    LOCAL CONST Robtarget Tr_meulage_bavure_258 := [[-0.894256591796875,91.7996015625,80.2160234375],[0.00347787918573702,-0.00302620431421481,0.656413988017704,-0.754386785925172],[0,0,0,0],[8.999999E+09,8.999999E+09,8.999999E+09,8.999999E+09,8.999999E+09,8.999999E+09]];
    LOCAL CONST Robtarget Tr_meulage_bavure_259 := [[-3.09170532226563,91.8315234375,80.2122734375],[0.00491374660901085,-0.00426989771840249,0.655908883103524,-0.754812003172727],[0,0,0,0],[8.999999E+09,8.999999E+09,8.999999E+09,8.999999E+09,8.999999E+09,8.999999E+09]];
    LOCAL CONST Robtarget Tr_meulage_bavure_260 := [[-8.3219912109375,91.974546875,80.1954765625],[0.00744982146467277,-0.00646558456435395,0.655423726856519,-0.755196950900821],[0,0,0,0],[8.999999E+09,8.999999E+09,8.999999E+09,8.999999E+09,8.999999E+09,8.999999E+09]];
    LOCAL CONST Robtarget Tr_meulage_bavure_261 := [[-9.6864931640625,91.992796875,80.193328125],[0.0113222387628506,-0.00981492756750365,0.654945437900396,-0.755527595445528],[0,0,0,0],[8.999999E+09,8.999999E+09,8.999999E+09,8.999999E+09,8.999999E+09,8.999999E+09]];
    LOCAL CONST Robtarget Tr_meulage_bavure_262 := [[-20.53646875,92.018953125,80.1902578125],[0.0166484079195255,-0.0144163975754932,0.65445477578378,-0.755780354632543],[0,0,0,0],[8.999999E+09,8.999999E+09,8.999999E+09,8.999999E+09,8.999999E+09,8.999999E+09]];
    LOCAL CONST Robtarget Tr_meulage_bavure_263 := [[-23.421142578125,92.016859375,80.1905],[0.0234300908490705,-0.020268509523459,0.653923705596549,-0.755925926016153],[0,0,0,0],[8.999999E+09,8.999999E+09,8.999999E+09,8.999999E+09,8.999999E+09,8.999999E+09]];
    LOCAL CONST Robtarget Tr_meulage_bavure_264 := [[-24.027587890625,92.04446875,80.1872578125],[0.0314797870413223,-0.0272072091200353,0.65333054540363,-0.755928560925123],[0,0,0,0],[8.999999E+09,8.999999E+09,8.999999E+09,8.999999E+09,8.999999E+09,8.999999E+09]];
    LOCAL CONST Robtarget Tr_meulage_bavure_265 := [[-26.45446875,92.1919921875,80.1699296875],[0.0404076636865339,-0.0348943430759381,0.652653550089562,-0.755773080423077],[0,0,0,0],[8.999999E+09,8.999999E+09,8.999999E+09,8.999999E+09,8.999999E+09,8.999999E+09]];
    LOCAL CONST Robtarget Tr_meulage_bavure_266 := [[-29.448517578125,92.303890625,80.15678125],[0.0496986305677145,-0.0428854622432543,0.651895870964166,-0.755461883001219],[0,0,0,0],[8.999999E+09,8.999999E+09,8.999999E+09,8.999999E+09,8.999999E+09,8.999999E+09]];
    LOCAL CONST Robtarget Tr_meulage_bavure_267 := [[-31.056060546875,92.1032109375,80.180359375],[0.0587225353541234,-0.0506383751390462,0.651088055954158,-0.755030967708409],[0,0,0,0],[8.999999E+09,8.999999E+09,8.999999E+09,8.999999E+09,8.999999E+09,8.999999E+09]];
    LOCAL CONST Robtarget Tr_meulage_bavure_268 := [[-35.77227734375,91.4953671875,80.251765625],[0.0668827998283126,-0.0576408748993466,0.650281395904972,-0.754545112480257],[0,0,0,0],[8.999999E+09,8.999999E+09,8.999999E+09,8.999999E+09,8.999999E+09,8.999999E+09]];
    LOCAL CONST Robtarget Tr_meulage_bavure_269 := [[-37.007875,91.1575078125,80.291453125],[0.0736958342973869,-0.0634793616298069,0.649541115383601,-0.754079328771524],[0,0,0,0],[8.999999E+09,8.999999E+09,8.999999E+09,8.999999E+09,8.999999E+09,8.999999E+09]];
    LOCAL CONST Robtarget Tr_meulage_bavure_270 := [[-38.72647265625,90.3674296875,80.384265625],[0.0789467515956599,-0.0679716715014017,0.648916433938356,-0.753694052020133],[0,0,0,0],[8.999999E+09,8.999999E+09,8.999999E+09,8.999999E+09,8.999999E+09,8.999999E+09]];
    LOCAL CONST Robtarget Tr_meulage_bavure_271 := [[-42.73101953125,88.3123828125,80.6256796875],[0.0827631719069685,-0.0712303856006982,0.648423147243865,-0.753408197235359],[0,0,0,0],[8.999999E+09,8.999999E+09,8.999999E+09,8.999999E+09,8.999999E+09,8.999999E+09]];
    LOCAL CONST Robtarget Tr_meulage_bavure_272 := [[-44.1032109375,87.88778125,80.6755546875],[0.0855847486840602,-0.0736356000993471,0.648035678832561,-0.753195066467325],[0,0,0,0],[8.999999E+09,8.999999E+09,8.999999E+09,8.999999E+09,8.999999E+09,8.999999E+09]];
    LOCAL CONST Robtarget Tr_meulage_bavure_273 := [[-46.86541796875,86.68584375,80.81675],[0.0882152360556618,-0.0758798732341398,0.647682492084163,-0.752972580120461],[0,0,0,0],[8.999999E+09,8.999999E+09,8.999999E+09,8.999999E+09,8.999999E+09,8.999999E+09]];
    LOCAL CONST Robtarget Tr_meulage_bavure_274 := [[-49.034421875,86.5238125,80.8357890625],[0.0916871696125905,-0.0788508623278929,0.647253511204557,-0.752621350130298],[0,0,0,0],[8.999999E+09,8.999999E+09,8.999999E+09,8.999999E+09,8.999999E+09,8.999999E+09]];
    LOCAL CONST Robtarget Tr_meulage_bavure_275 := [[-53.57986328125,85.9536640625,80.902765625],[0.0972011976752642,-0.0835810818582939,0.646606172682112,-0.751975124173189],[0,0,0,0],[8.999999E+09,8.999999E+09,8.999999E+09,8.999999E+09,8.999999E+09,8.999999E+09]];
    LOCAL CONST Robtarget Tr_meulage_bavure_276 := [[-59.01324609375,86.3367734375,80.8577578125],[0.106067029700948,-0.0911960835370439,0.645540805269948,-0.750806318759605],[0,0,0,0],[8.999999E+09,8.999999E+09,8.999999E+09,8.999999E+09,8.999999E+09,8.999999E+09]];
    LOCAL CONST Robtarget Tr_meulage_bavure_277 := [[-61.2616875,86.3511640625,80.8560703125],[0.119501918726964,-0.10274216646515,0.643784911960041,-0.748801926936105],[0,0,0,0],[8.999999E+09,8.999999E+09,8.999999E+09,8.999999E+09,8.999999E+09,8.999999E+09]];
    LOCAL CONST Robtarget Tr_meulage_bavure_278 := [[-69.158140625,86.6093671875,80.825734375],[0.13852846594866,-0.119099643075277,0.640958292885336,-0.745518347140276],[0,0,0,0],[8.999999E+09,8.999999E+09,8.999999E+09,8.999999E+09,8.999999E+09,8.999999E+09]];
    LOCAL CONST Robtarget Tr_meulage_bavure_279 := [[-70.97525,86.6130703125,80.8253046875],[0.163876976589741,-0.140896368891585,0.636531382818664,-0.740351503317128],[0,0,0,0],[8.999999E+09,8.999999E+09,8.999999E+09,8.999999E+09,8.999999E+09,8.999999E+09]];
    LOCAL CONST Robtarget Tr_meulage_bavure_280 := [[-73.90365625,86.3363203125,80.8578125],[0.195657464814664,-0.168229660305411,0.629881023434704,-0.732575480187997],[0,0,0,0],[8.999999E+09,8.999999E+09,8.999999E+09,8.999999E+09,8.999999E+09,8.999999E+09]];
    LOCAL CONST Robtarget Tr_meulage_bavure_281 := [[-75.0881328125,86.0497421875,80.8914765625],[0.233090996505808,-0.200432374900431,0.620418372993561,-0.721509870266323],[0,0,0,0],[8.999999E+09,8.999999E+09,8.999999E+09,8.999999E+09,8.999999E+09,8.999999E+09]];
    LOCAL CONST Robtarget Tr_meulage_bavure_282 := [[-77.5441015625,85.085125,81.004796875],[0.274367163117045,-0.235949651903377,0.607840699423548,-0.706809808713824],[0,0,0,0],[8.999999E+09,8.999999E+09,8.999999E+09,8.999999E+09,8.999999E+09,8.999999E+09]];
    LOCAL CONST Robtarget Tr_meulage_bavure_283 := [[-78.4228515625,84.0872265625,81.1220234375],[0.316761155122173,-0.272440578103132,0.592433930974092,-0.688810960597378],[0,0,0,0],[8.999999E+09,8.999999E+09,8.999999E+09,8.999999E+09,8.999999E+09,8.999999E+09]];
    LOCAL CONST Robtarget Tr_meulage_bavure_284 := [[-79.9829375,82.004625,81.366671875],[0.357317508371397,-0.307363032722583,0.575147348147079,-0.668623729945487],[0,0,0,0],[8.999999E+09,8.999999E+09,8.999999E+09,8.999999E+09,8.999999E+09,8.999999E+09]];
    LOCAL CONST Robtarget Tr_meulage_bavure_285 := [[-80.3374296875,79.783875,81.627546875],[0.393613708380539,-0.33863296716412,0.557372094713365,-0.647867509726626],[0,0,0,0],[8.999999E+09,8.999999E+09,8.999999E+09,8.999999E+09,8.999999E+09,8.999999E+09]];
    LOCAL CONST Robtarget Tr_meulage_bavure_286 := [[-80.412265625,79.58646875,81.6507421875],[0.424278534863153,-0.365066131411498,0.540492222763307,-0.628158102457493],[0,0,0,0],[8.999999E+09,8.999999E+09,8.999999E+09,8.999999E+09,8.999999E+09,8.999999E+09]];
    LOCAL CONST Robtarget Tr_meulage_bavure_287 := [[-80.42434375,79.4588359375,81.665734375],[0.448961364969328,-0.38635898724885,0.525548437863281,-0.610703909596448],[0,0,0,0],[8.999999E+09,8.999999E+09,8.999999E+09,8.999999E+09,8.999999E+09,8.999999E+09]];
    LOCAL CONST Robtarget Tr_meulage_bavure_288 := [[-80.630734375,75.5483203125,82.125109375],[0.467989879490766,-0.402790192772944,0.513130058558757,-0.596190469819536],[0,0,0,0],[8.999999E+09,8.999999E+09,8.999999E+09,8.999999E+09,8.999999E+09,8.999999E+09]];
    LOCAL CONST Robtarget Tr_meulage_bavure_289 := [[-80.5011015625,72.5830859375,82.4734453125],[0.482071863396728,-0.414965340552088,0.503399466828588,-0.584807200244994],[0,0,0,0],[8.999999E+09,8.999999E+09,8.999999E+09,8.999999E+09,8.999999E+09,8.999999E+09]];
    LOCAL CONST Robtarget Tr_meulage_bavure_290 := [[-80.316984375,68.9543203125,82.8997265625],[0.49206179036456,-0.423611707299164,0.4962002859683,-0.576379729091237],[0,0,0,0],[8.999999E+09,8.999999E+09,8.999999E+09,8.999999E+09,8.999999E+09,8.999999E+09]];
    LOCAL CONST Robtarget Tr_meulage_bavure_291 := [[-80.258484375,65.9367109375,83.25421875],[0.498791013906897,-0.429448562893376,0.491208022376699,-0.570522685813033],[0,0,0,0],[8.999999E+09,8.999999E+09,8.999999E+09,8.999999E+09,8.999999E+09,8.999999E+09]];
    LOCAL CONST Robtarget Tr_meulage_bavure_292 := [[-80.1468203125,54.898046875,84.5509609375],[0.503007913688158,-0.43312019155188,0.488021045124207,-0.566767499026741],[0,0,0,0],[8.999999E+09,8.999999E+09,8.999999E+09,8.999999E+09,8.999999E+09,8.999999E+09]];
    LOCAL CONST Robtarget Tr_meulage_bavure_293 := [[-80.2864375,48.8831328125,85.2575546875],[0.505447763460853,-0.435251867230867,0.486156431674502,-0.564562037712402],[0,0,0,0],[8.999999E+09,8.999999E+09,8.999999E+09,8.999999E+09,8.999999E+09,8.999999E+09]];
    LOCAL CONST Robtarget Tr_meulage_bavure_294 := [[-80.335140625,46.1458203125,85.579109375],[0.50671707315682,-0.436369685524733,0.485181965999149,-0.56339840716462],[0,0,0,0],[8.999999E+09,8.999999E+09,8.999999E+09,8.999999E+09,8.999999E+09,8.999999E+09]];
    LOCAL CONST Robtarget Tr_meulage_bavure_295 := [[-80.3631015625,45.63105078125,85.6395859375],[0.507275210539017,-0.436864892405638,0.484752927928074,-0.56288144881597],[0,0,0,0],[8.999999E+09,8.999999E+09,8.999999E+09,8.999999E+09,8.999999E+09,8.999999E+09]];
    LOCAL CONST Robtarget Tr_meulage_bavure_296 := [[-80.6398046875,44.21337109375,85.806125],[0.507430369539302,-0.437006893390196,0.484634589770416,-0.562733249059194],[0,0,0,0],[8.999999E+09,8.999999E+09,8.999999E+09,8.999999E+09,8.999999E+09,8.999999E+09]];
    !
    !Declaration des points de tronconnage

    !
    !Cycle
    LOCAL PROC Cycle()
        !
        Prise;
        !
        Meulage;
        !
        !
        Depose;
        !
    ENDPROC

    !Trajectoire de prise de la pièce
    LOCAL PROC PRISE()

		!
        !Trigger localisation
        LocalisationPieceTable 703 \model:=1;
        !
        !Approche
		MoveJ Reltool(PicKPosition,0,0,-100),V1000,Z0,Tool_Prehenseur1 \Wobj:=Wobj_vision;
		MoveL Reltool(PicKPosition,0,0,-50),V500,Z0,Tool_Prehenseur1 \Wobj:=Wobj_vision;
		MoveL Reltool(PicKPosition,0,0,-10),V200,Z0,Tool_Prehenseur1 \Wobj:=Wobj_vision;
		MoveL PicKPosition,V100,Fine,Tool_Prehenseur1 \Wobj:=Wobj_vision;

        !Fermeture pince
		Gripper_Close;
        !
		MoveL Reltool(PicKPosition,0,0,-100),V500,Z0,Tool_Prehenseur1 \Wobj:=Wobj_vision;

        !Trigger relocalisation
		LocalisationPiecePrehenseur 703 \model:=1,Ref;
        !
        PEO;
        !
    ENDPROC

    !Trajectoire de tronconnage
    LOCAL PROC Tronconnage()
        !
        !StartMotor1();
        !
        ConfJ \Off;
        ConfL \Off;


    ENDPROC


    !Trajectoire de meulage
    LOCAL PROC Meulage()
        !
        !StartMotor2();
        !

        ConfJ \Off;
        ConfL \Off;


        !---------- Meulage zone : 1 ------------

        !Approche PLAN

        Go_to_Meulage_Plan;
		Tool := ToolOffset(Tool_M1_D500_S0 \Z);

        !
        !Approche
        MoveJ Reltool(Tr_meulage_motif_1_0,0,0,-200),V1000,Z0,Tool \Wobj:=Wobj_Part_0;
        MoveL Reltool(Tr_meulage_motif_1_0,0,0,-100),V500,Z0,Tool \Wobj:=Wobj_Part_0;
        MoveL Reltool(Tr_meulage_motif_1_0,0,0,-10),V100,Z0,Tool \Wobj:=Wobj_Part_0;
        !
        !Trajectoire
        Movel Tr_meulage_motif_1_0,VitesseLente,Z0,Tool \Wobj:=Wobj_Part_0;
        Movel Tr_meulage_motif_1_1,VitesseLente,Z0,Tool \Wobj:=Wobj_Part_0;
        Movel Tr_meulage_motif_1_2,VitesseLente,Z0,Tool \Wobj:=Wobj_Part_0;
        Movel Tr_meulage_motif_1_3,VitesseLente,Z0,Tool \Wobj:=Wobj_Part_0;
        Movel Tr_meulage_motif_1_4,VitesseLente,Z0,Tool \Wobj:=Wobj_Part_0;
        Movel Tr_meulage_motif_1_5,VitesseLente,Z0,Tool \Wobj:=Wobj_Part_0;
        Movel Tr_meulage_motif_1_6,VitesseLente,Z0,Tool \Wobj:=Wobj_Part_0;
        Movel Tr_meulage_motif_1_7,VitesseLente,Z0,Tool \Wobj:=Wobj_Part_0;
        Movel Tr_meulage_motif_1_8,VitesseLente,Z0,Tool \Wobj:=Wobj_Part_0;
        Movel Tr_meulage_motif_1_9,VitesseLente,Z0,Tool \Wobj:=Wobj_Part_0;
        Movel Tr_meulage_motif_1_10,VitesseLente,Z0,Tool \Wobj:=Wobj_Part_0;
        Movel Tr_meulage_motif_1_11,VitesseLente,Z0,Tool \Wobj:=Wobj_Part_0;
        Movel Tr_meulage_motif_1_12,VitesseLente,Z0,Tool \Wobj:=Wobj_Part_0;
        Movel Tr_meulage_motif_1_13,VitesseLente,Z0,Tool \Wobj:=Wobj_Part_0;
        Movel Tr_meulage_motif_1_14,VitesseLente,Z0,Tool \Wobj:=Wobj_Part_0;
        Movel Tr_meulage_motif_1_15,VitesseLente,Z0,Tool \Wobj:=Wobj_Part_0;
        Movel Tr_meulage_motif_1_16,VitesseLente,Z0,Tool \Wobj:=Wobj_Part_0;
        Movel Tr_meulage_motif_1_17,VitesseLente,Z0,Tool \Wobj:=Wobj_Part_0;
        Movel Tr_meulage_motif_1_18,VitesseLente,Z0,Tool \Wobj:=Wobj_Part_0;
        Movel Tr_meulage_motif_1_19,VitesseLente,Z0,Tool \Wobj:=Wobj_Part_0;
        Movel Tr_meulage_motif_1_20,VitesseLente,Z0,Tool \Wobj:=Wobj_Part_0;
        Movel Tr_meulage_motif_1_21,VitesseLente,Z0,Tool \Wobj:=Wobj_Part_0;
        Movel Tr_meulage_motif_1_22,VitesseLente,Z0,Tool \Wobj:=Wobj_Part_0;
        Movel Tr_meulage_motif_1_23,VitesseLente,Z0,Tool \Wobj:=Wobj_Part_0;
        Movel Tr_meulage_motif_1_24,VitesseLente,Z0,Tool \Wobj:=Wobj_Part_0;
        Movel Tr_meulage_motif_1_25,VitesseLente,Z0,Tool \Wobj:=Wobj_Part_0;
        Movel Tr_meulage_motif_1_26,VitesseLente,Z0,Tool \Wobj:=Wobj_Part_0;
        Movel Tr_meulage_motif_1_27,VitesseLente,Z0,Tool \Wobj:=Wobj_Part_0;
        Movel Tr_meulage_motif_1_28,VitesseLente,Z0,Tool \Wobj:=Wobj_Part_0;
        Movel Tr_meulage_motif_1_29,VitesseLente,Z0,Tool \Wobj:=Wobj_Part_0;
        Movel Tr_meulage_motif_1_30,VitesseLente,Z0,Tool \Wobj:=Wobj_Part_0;
        Movel Tr_meulage_motif_1_31,VitesseLente,Z0,Tool \Wobj:=Wobj_Part_0;
        Movel Tr_meulage_motif_1_32,VitesseLente,Z0,Tool \Wobj:=Wobj_Part_0;
        Movel Tr_meulage_motif_1_33,VitesseLente,Z0,Tool \Wobj:=Wobj_Part_0;
        Movel Tr_meulage_motif_1_34,VitesseLente,Z0,Tool \Wobj:=Wobj_Part_0;
        Movel Tr_meulage_motif_1_35,VitesseLente,Z0,Tool \Wobj:=Wobj_Part_0;
        Movel Tr_meulage_motif_1_36,VitesseLente,Z0,Tool \Wobj:=Wobj_Part_0;
        Movel Tr_meulage_motif_1_37,VitesseLente,Z0,Tool \Wobj:=Wobj_Part_0;
        Movel Tr_meulage_motif_1_38,VitesseLente,Z0,Tool \Wobj:=Wobj_Part_0;
        Movel Tr_meulage_motif_1_39,VitesseLente,Z0,Tool \Wobj:=Wobj_Part_0;
        Movel Tr_meulage_motif_1_40,VitesseLente,Z0,Tool \Wobj:=Wobj_Part_0;
        Movel Tr_meulage_motif_1_41,VitesseLente,Z0,Tool \Wobj:=Wobj_Part_0;
        Movel Tr_meulage_motif_1_42,VitesseLente,Z0,Tool \Wobj:=Wobj_Part_0;
        Movel Tr_meulage_motif_1_43,VitesseLente,Z0,Tool \Wobj:=Wobj_Part_0;
        Movel Tr_meulage_motif_1_44,VitesseLente,Z0,Tool \Wobj:=Wobj_Part_0;
        Movel Tr_meulage_motif_1_45,VitesseLente,Z0,Tool \Wobj:=Wobj_Part_0;
        Movel Tr_meulage_motif_1_46,VitesseLente,Z0,Tool \Wobj:=Wobj_Part_0;
        Movel Tr_meulage_motif_1_47,VitesseLente,Z0,Tool \Wobj:=Wobj_Part_0;
        Movel Tr_meulage_motif_1_48,VitesseLente,Z0,Tool \Wobj:=Wobj_Part_0;
        Movel Tr_meulage_motif_1_49,VitesseLente,Z0,Tool \Wobj:=Wobj_Part_0;
        Movel Tr_meulage_motif_1_50,VitesseLente,Z0,Tool \Wobj:=Wobj_Part_0;
        Movel Tr_meulage_motif_1_51,VitesseLente,Z0,Tool \Wobj:=Wobj_Part_0;
        Movel Tr_meulage_motif_1_52,VitesseLente,Z0,Tool \Wobj:=Wobj_Part_0;
        Movel Tr_meulage_motif_1_53,VitesseLente,Z0,Tool \Wobj:=Wobj_Part_0;
        Movel Tr_meulage_motif_1_54,VitesseLente,Z0,Tool \Wobj:=Wobj_Part_0;
        Movel Tr_meulage_motif_1_55,VitesseLente,Z0,Tool \Wobj:=Wobj_Part_0;
        Movel Tr_meulage_motif_1_56,VitesseLente,Z0,Tool \Wobj:=Wobj_Part_0;
        Movel Tr_meulage_motif_1_57,VitesseLente,Z0,Tool \Wobj:=Wobj_Part_0;
        Movel Tr_meulage_motif_1_58,VitesseLente,Z0,Tool \Wobj:=Wobj_Part_0;
        Movel Tr_meulage_motif_1_59,VitesseLente,Z0,Tool \Wobj:=Wobj_Part_0;
        Movel Tr_meulage_motif_1_60,VitesseLente,Z0,Tool \Wobj:=Wobj_Part_0;
        Movel Tr_meulage_motif_1_61,VitesseLente,Z0,Tool \Wobj:=Wobj_Part_0;
        Movel Tr_meulage_motif_1_62,VitesseLente,Z0,Tool \Wobj:=Wobj_Part_0;
        Movel Tr_meulage_motif_1_63,VitesseLente,Z0,Tool \Wobj:=Wobj_Part_0;
        Movel Tr_meulage_motif_1_64,VitesseLente,Z0,Tool \Wobj:=Wobj_Part_0;
        Movel Tr_meulage_motif_1_65,VitesseLente,Z0,Tool \Wobj:=Wobj_Part_0;
        Movel Tr_meulage_motif_1_66,VitesseLente,Z0,Tool \Wobj:=Wobj_Part_0;
        Movel Tr_meulage_motif_1_67,VitesseLente,Z0,Tool \Wobj:=Wobj_Part_0;
        Movel Tr_meulage_motif_1_68,VitesseLente,Z0,Tool \Wobj:=Wobj_Part_0;
        Movel Tr_meulage_motif_1_69,VitesseLente,Z0,Tool \Wobj:=Wobj_Part_0;
        Movel Tr_meulage_motif_1_70,VitesseLente,Z0,Tool \Wobj:=Wobj_Part_0;
        Movel Tr_meulage_motif_1_71,VitesseLente,Z0,Tool \Wobj:=Wobj_Part_0;
        Movel Tr_meulage_motif_1_72,VitesseLente,Z0,Tool \Wobj:=Wobj_Part_0;
        Movel Tr_meulage_motif_1_73,VitesseLente,Z0,Tool \Wobj:=Wobj_Part_0;
        Movel Tr_meulage_motif_1_74,VitesseLente,Z0,Tool \Wobj:=Wobj_Part_0;
        Movel Tr_meulage_motif_1_75,VitesseLente,Z0,Tool \Wobj:=Wobj_Part_0;
        Movel Tr_meulage_motif_1_76,VitesseLente,Z0,Tool \Wobj:=Wobj_Part_0;
        Movel Tr_meulage_motif_1_77,VitesseLente,Z0,Tool \Wobj:=Wobj_Part_0;
        Movel Tr_meulage_motif_1_78,VitesseLente,Z0,Tool \Wobj:=Wobj_Part_0;
        Movel Tr_meulage_motif_1_79,VitesseLente,Z0,Tool \Wobj:=Wobj_Part_0;
        Movel Tr_meulage_motif_1_80,VitesseLente,Z0,Tool \Wobj:=Wobj_Part_0;
        Movel Tr_meulage_motif_1_81,VitesseLente,Z0,Tool \Wobj:=Wobj_Part_0;
        Movel Tr_meulage_motif_1_82,VitesseLente,Z0,Tool \Wobj:=Wobj_Part_0;
        Movel Tr_meulage_motif_1_83,VitesseLente,Z0,Tool \Wobj:=Wobj_Part_0;
        Movel Tr_meulage_motif_1_84,VitesseLente,Z0,Tool \Wobj:=Wobj_Part_0;
        Movel Tr_meulage_motif_1_85,VitesseLente,Z0,Tool \Wobj:=Wobj_Part_0;
        Movel Tr_meulage_motif_1_86,VitesseLente,Z0,Tool \Wobj:=Wobj_Part_0;
        Movel Tr_meulage_motif_1_87,VitesseLente,Z0,Tool \Wobj:=Wobj_Part_0;
        Movel Tr_meulage_motif_1_88,VitesseLente,Z0,Tool \Wobj:=Wobj_Part_0;
        Movel Tr_meulage_motif_1_89,VitesseLente,Z0,Tool \Wobj:=Wobj_Part_0;
        Movel Tr_meulage_motif_1_90,VitesseLente,Z0,Tool \Wobj:=Wobj_Part_0;
        Movel Tr_meulage_motif_1_91,VitesseLente,Z0,Tool \Wobj:=Wobj_Part_0;
        Movel Tr_meulage_motif_1_92,VitesseLente,Z0,Tool \Wobj:=Wobj_Part_0;
        Movel Tr_meulage_motif_1_93,VitesseLente,Z0,Tool \Wobj:=Wobj_Part_0;
        Movel Tr_meulage_motif_1_94,VitesseLente,Z0,Tool \Wobj:=Wobj_Part_0;
        Movel Tr_meulage_motif_1_95,VitesseLente,Z0,Tool \Wobj:=Wobj_Part_0;
        Movel Tr_meulage_motif_1_96,VitesseLente,Z0,Tool \Wobj:=Wobj_Part_0;
        Movel Tr_meulage_motif_1_97,VitesseLente,Z0,Tool \Wobj:=Wobj_Part_0;
        Movel Tr_meulage_motif_1_98,VitesseLente,Z0,Tool \Wobj:=Wobj_Part_0;
        Movel Tr_meulage_motif_1_99,VitesseLente,Z0,Tool \Wobj:=Wobj_Part_0;
        Movel Tr_meulage_motif_1_100,VitesseLente,Z0,Tool \Wobj:=Wobj_Part_0;
        Movel Tr_meulage_motif_1_101,VitesseLente,Z0,Tool \Wobj:=Wobj_Part_0;
        Movel Tr_meulage_motif_1_102,VitesseLente,Z0,Tool \Wobj:=Wobj_Part_0;
        Movel Tr_meulage_motif_1_103,VitesseLente,Z0,Tool \Wobj:=Wobj_Part_0;
        Movel Tr_meulage_motif_1_104,VitesseLente,Z0,Tool \Wobj:=Wobj_Part_0;
        Movel Tr_meulage_motif_1_105,VitesseLente,Z0,Tool \Wobj:=Wobj_Part_0;
        Movel Tr_meulage_motif_1_106,VitesseLente,Z0,Tool \Wobj:=Wobj_Part_0;
        Movel Tr_meulage_motif_1_107,VitesseLente,Z0,Tool \Wobj:=Wobj_Part_0;
        Movel Tr_meulage_motif_1_108,VitesseLente,Z0,Tool \Wobj:=Wobj_Part_0;
        Movel Tr_meulage_motif_1_109,VitesseLente,Z0,Tool \Wobj:=Wobj_Part_0;
        Movel Tr_meulage_motif_1_110,VitesseLente,Z0,Tool \Wobj:=Wobj_Part_0;
        Movel Tr_meulage_motif_1_111,VitesseLente,Z0,Tool \Wobj:=Wobj_Part_0;
        Movel Tr_meulage_motif_1_112,VitesseLente,Z0,Tool \Wobj:=Wobj_Part_0;
        Movel Tr_meulage_motif_1_113,VitesseLente,Z0,Tool \Wobj:=Wobj_Part_0;
        Movel Tr_meulage_motif_1_114,VitesseLente,Z0,Tool \Wobj:=Wobj_Part_0;
        Movel Tr_meulage_motif_1_115,VitesseLente,Z0,Tool \Wobj:=Wobj_Part_0;
        !
        !Degagement
        MoveL Reltool(Tr_meulage_motif_1_115,0,0,-10),V100,Z0,Tool \Wobj:=Wobj_Part_0;
        MoveL Reltool(Tr_meulage_motif_1_115,0,0,-100),V500,Z0,Tool \Wobj:=Wobj_Part_0;
        MoveJ Reltool(Tr_meulage_motif_1_115,0,0,-200),V1000,Z0,Tool \Wobj:=Wobj_Part_0;


        Go_to_Meulage_Plan;
        !
        !

        !---------- Meulage zone : 2 ------------

        !Approche PLAN

        Go_to_Meulage_Plan;
		Tool := ToolOffset(Tool_M1_D500_S0 \Z);

        !
        !Approche
        MoveJ Reltool(Tr_meulage_bavure_0,0,0,-200),V1000,Z0,Tool \Wobj:=Wobj_Part_0;
        MoveL Reltool(Tr_meulage_bavure_0,0,0,-100),V500,Z0,Tool \Wobj:=Wobj_Part_0;
        MoveL Reltool(Tr_meulage_bavure_0,0,0,-10),V100,Z0,Tool \Wobj:=Wobj_Part_0;
        !
        !Trajectoire
        Movel Tr_meulage_bavure_0,VitesseRapide,Z0,Tool \Wobj:=Wobj_Part_0;
        Movel Tr_meulage_bavure_1,VitesseRapide,Z0,Tool \Wobj:=Wobj_Part_0;
        Movel Tr_meulage_bavure_2,VitesseRapide,Z0,Tool \Wobj:=Wobj_Part_0;
        Movel Tr_meulage_bavure_3,VitesseRapide,Z0,Tool \Wobj:=Wobj_Part_0;
        Movel Tr_meulage_bavure_4,VitesseRapide,Z0,Tool \Wobj:=Wobj_Part_0;
        Movel Tr_meulage_bavure_5,VitesseRapide,Z0,Tool \Wobj:=Wobj_Part_0;
        Movel Tr_meulage_bavure_6,VitesseRapide,Z0,Tool \Wobj:=Wobj_Part_0;
        Movel Tr_meulage_bavure_7,VitesseRapide,Z0,Tool \Wobj:=Wobj_Part_0;
        Movel Tr_meulage_bavure_8,VitesseRapide,Z0,Tool \Wobj:=Wobj_Part_0;
        Movel Tr_meulage_bavure_9,VitesseRapide,Z0,Tool \Wobj:=Wobj_Part_0;
        Movel Tr_meulage_bavure_10,VitesseRapide,Z0,Tool \Wobj:=Wobj_Part_0;
        Movel Tr_meulage_bavure_11,VitesseRapide,Z0,Tool \Wobj:=Wobj_Part_0;
        Movel Tr_meulage_bavure_12,VitesseRapide,Z0,Tool \Wobj:=Wobj_Part_0;
        Movel Tr_meulage_bavure_13,VitesseRapide,Z0,Tool \Wobj:=Wobj_Part_0;
        Movel Tr_meulage_bavure_14,VitesseRapide,Z0,Tool \Wobj:=Wobj_Part_0;
        Movel Tr_meulage_bavure_15,VitesseRapide,Z0,Tool \Wobj:=Wobj_Part_0;
        Movel Tr_meulage_bavure_16,VitesseRapide,Z0,Tool \Wobj:=Wobj_Part_0;
        Movel Tr_meulage_bavure_17,VitesseRapide,Z0,Tool \Wobj:=Wobj_Part_0;
        Movel Tr_meulage_bavure_18,VitesseRapide,Z0,Tool \Wobj:=Wobj_Part_0;
        Movel Tr_meulage_bavure_19,VitesseRapide,Z0,Tool \Wobj:=Wobj_Part_0;
        Movel Tr_meulage_bavure_20,VitesseRapide,Z0,Tool \Wobj:=Wobj_Part_0;
        Movel Tr_meulage_bavure_21,VitesseRapide,Z0,Tool \Wobj:=Wobj_Part_0;
        Movel Tr_meulage_bavure_22,VitesseRapide,Z0,Tool \Wobj:=Wobj_Part_0;
        Movel Tr_meulage_bavure_23,VitesseRapide,Z0,Tool \Wobj:=Wobj_Part_0;
        Movel Tr_meulage_bavure_24,VitesseRapide,Z0,Tool \Wobj:=Wobj_Part_0;
        Movel Tr_meulage_bavure_25,VitesseRapide,Z0,Tool \Wobj:=Wobj_Part_0;
        Movel Tr_meulage_bavure_26,VitesseRapide,Z0,Tool \Wobj:=Wobj_Part_0;
        Movel Tr_meulage_bavure_27,VitesseRapide,Z0,Tool \Wobj:=Wobj_Part_0;
        Movel Tr_meulage_bavure_28,VitesseRapide,Z0,Tool \Wobj:=Wobj_Part_0;
        Movel Tr_meulage_bavure_29,VitesseRapide,Z0,Tool \Wobj:=Wobj_Part_0;
        Movel Tr_meulage_bavure_30,VitesseRapide,Z0,Tool \Wobj:=Wobj_Part_0;
        Movel Tr_meulage_bavure_31,VitesseRapide,Z0,Tool \Wobj:=Wobj_Part_0;
        Movel Tr_meulage_bavure_32,VitesseRapide,Z0,Tool \Wobj:=Wobj_Part_0;
        Movel Tr_meulage_bavure_33,VitesseRapide,Z0,Tool \Wobj:=Wobj_Part_0;
        Movel Tr_meulage_bavure_34,VitesseRapide,Z0,Tool \Wobj:=Wobj_Part_0;
        Movel Tr_meulage_bavure_35,VitesseRapide,Z0,Tool \Wobj:=Wobj_Part_0;
        Movel Tr_meulage_bavure_36,VitesseRapide,Z0,Tool \Wobj:=Wobj_Part_0;
        Movel Tr_meulage_bavure_37,VitesseRapide,Z0,Tool \Wobj:=Wobj_Part_0;
        Movel Tr_meulage_bavure_38,VitesseRapide,Z0,Tool \Wobj:=Wobj_Part_0;
        Movel Tr_meulage_bavure_39,VitesseRapide,Z0,Tool \Wobj:=Wobj_Part_0;
        Movel Tr_meulage_bavure_40,VitesseRapide,Z0,Tool \Wobj:=Wobj_Part_0;
        Movel Tr_meulage_bavure_41,VitesseRapide,Z0,Tool \Wobj:=Wobj_Part_0;
        Movel Tr_meulage_bavure_42,VitesseRapide,Z0,Tool \Wobj:=Wobj_Part_0;
        Movel Tr_meulage_bavure_43,VitesseRapide,Z0,Tool \Wobj:=Wobj_Part_0;
        Movel Tr_meulage_bavure_44,VitesseRapide,Z0,Tool \Wobj:=Wobj_Part_0;
        Movel Tr_meulage_bavure_45,VitesseRapide,Z0,Tool \Wobj:=Wobj_Part_0;
        Movel Tr_meulage_bavure_46,VitesseRapide,Z0,Tool \Wobj:=Wobj_Part_0;
        Movel Tr_meulage_bavure_47,VitesseRapide,Z0,Tool \Wobj:=Wobj_Part_0;
        Movel Tr_meulage_bavure_48,VitesseRapide,Z0,Tool \Wobj:=Wobj_Part_0;
        Movel Tr_meulage_bavure_49,VitesseRapide,Z0,Tool \Wobj:=Wobj_Part_0;
        Movel Tr_meulage_bavure_50,VitesseRapide,Z0,Tool \Wobj:=Wobj_Part_0;
        Movel Tr_meulage_bavure_51,VitesseRapide,Z0,Tool \Wobj:=Wobj_Part_0;
        Movel Tr_meulage_bavure_52,VitesseRapide,Z0,Tool \Wobj:=Wobj_Part_0;
        Movel Tr_meulage_bavure_53,VitesseRapide,Z0,Tool \Wobj:=Wobj_Part_0;
        Movel Tr_meulage_bavure_54,VitesseRapide,Z0,Tool \Wobj:=Wobj_Part_0;
        Movel Tr_meulage_bavure_55,VitesseRapide,Z0,Tool \Wobj:=Wobj_Part_0;
        Movel Tr_meulage_bavure_56,VitesseRapide,Z0,Tool \Wobj:=Wobj_Part_0;
        Movel Tr_meulage_bavure_57,VitesseRapide,Z0,Tool \Wobj:=Wobj_Part_0;
        Movel Tr_meulage_bavure_58,VitesseRapide,Z0,Tool \Wobj:=Wobj_Part_0;
        Movel Tr_meulage_bavure_59,VitesseRapide,Z0,Tool \Wobj:=Wobj_Part_0;
        Movel Tr_meulage_bavure_60,VitesseRapide,Z0,Tool \Wobj:=Wobj_Part_0;
        Movel Tr_meulage_bavure_61,VitesseRapide,Z0,Tool \Wobj:=Wobj_Part_0;
        Movel Tr_meulage_bavure_62,VitesseRapide,Z0,Tool \Wobj:=Wobj_Part_0;
        Movel Tr_meulage_bavure_63,VitesseRapide,Z0,Tool \Wobj:=Wobj_Part_0;
        Movel Tr_meulage_bavure_64,VitesseRapide,Z0,Tool \Wobj:=Wobj_Part_0;
        Movel Tr_meulage_bavure_65,VitesseRapide,Z0,Tool \Wobj:=Wobj_Part_0;
        Movel Tr_meulage_bavure_66,VitesseRapide,Z0,Tool \Wobj:=Wobj_Part_0;
        Movel Tr_meulage_bavure_67,VitesseRapide,Z0,Tool \Wobj:=Wobj_Part_0;
        Movel Tr_meulage_bavure_68,VitesseRapide,Z0,Tool \Wobj:=Wobj_Part_0;
        Movel Tr_meulage_bavure_69,VitesseRapide,Z0,Tool \Wobj:=Wobj_Part_0;
        Movel Tr_meulage_bavure_70,VitesseRapide,Z0,Tool \Wobj:=Wobj_Part_0;
        Movel Tr_meulage_bavure_71,VitesseRapide,Z0,Tool \Wobj:=Wobj_Part_0;
        Movel Tr_meulage_bavure_72,VitesseRapide,Z0,Tool \Wobj:=Wobj_Part_0;
        Movel Tr_meulage_bavure_73,VitesseRapide,Z0,Tool \Wobj:=Wobj_Part_0;
        Movel Tr_meulage_bavure_74,VitesseRapide,Z0,Tool \Wobj:=Wobj_Part_0;
        Movel Tr_meulage_bavure_75,VitesseRapide,Z0,Tool \Wobj:=Wobj_Part_0;
        Movel Tr_meulage_bavure_76,VitesseRapide,Z0,Tool \Wobj:=Wobj_Part_0;
        Movel Tr_meulage_bavure_77,VitesseRapide,Z0,Tool \Wobj:=Wobj_Part_0;
        Movel Tr_meulage_bavure_78,VitesseRapide,Z0,Tool \Wobj:=Wobj_Part_0;
        Movel Tr_meulage_bavure_79,VitesseRapide,Z0,Tool \Wobj:=Wobj_Part_0;
        Movel Tr_meulage_bavure_80,VitesseRapide,Z0,Tool \Wobj:=Wobj_Part_0;
        Movel Tr_meulage_bavure_81,VitesseRapide,Z0,Tool \Wobj:=Wobj_Part_0;
        Movel Tr_meulage_bavure_82,VitesseRapide,Z0,Tool \Wobj:=Wobj_Part_0;
        Movel Tr_meulage_bavure_83,VitesseRapide,Z0,Tool \Wobj:=Wobj_Part_0;
        Movel Tr_meulage_bavure_84,VitesseRapide,Z0,Tool \Wobj:=Wobj_Part_0;
        Movel Tr_meulage_bavure_85,VitesseRapide,Z0,Tool \Wobj:=Wobj_Part_0;
        Movel Tr_meulage_bavure_86,VitesseRapide,Z0,Tool \Wobj:=Wobj_Part_0;
        Movel Tr_meulage_bavure_87,VitesseRapide,Z0,Tool \Wobj:=Wobj_Part_0;
        Movel Tr_meulage_bavure_88,VitesseRapide,Z0,Tool \Wobj:=Wobj_Part_0;
        Movel Tr_meulage_bavure_89,VitesseRapide,Z0,Tool \Wobj:=Wobj_Part_0;
        Movel Tr_meulage_bavure_90,VitesseRapide,Z0,Tool \Wobj:=Wobj_Part_0;
        Movel Tr_meulage_bavure_91,VitesseRapide,Z0,Tool \Wobj:=Wobj_Part_0;
        Movel Tr_meulage_bavure_92,VitesseRapide,Z0,Tool \Wobj:=Wobj_Part_0;
        Movel Tr_meulage_bavure_93,VitesseRapide,Z0,Tool \Wobj:=Wobj_Part_0;
        Movel Tr_meulage_bavure_94,VitesseRapide,Z0,Tool \Wobj:=Wobj_Part_0;
        Movel Tr_meulage_bavure_95,VitesseRapide,Z0,Tool \Wobj:=Wobj_Part_0;
        Movel Tr_meulage_bavure_96,VitesseRapide,Z0,Tool \Wobj:=Wobj_Part_0;
        Movel Tr_meulage_bavure_97,VitesseRapide,Z0,Tool \Wobj:=Wobj_Part_0;
        Movel Tr_meulage_bavure_98,VitesseRapide,Z0,Tool \Wobj:=Wobj_Part_0;
        Movel Tr_meulage_bavure_99,VitesseRapide,Z0,Tool \Wobj:=Wobj_Part_0;
        Movel Tr_meulage_bavure_100,VitesseRapide,Z0,Tool \Wobj:=Wobj_Part_0;
        Movel Tr_meulage_bavure_101,VitesseRapide,Z0,Tool \Wobj:=Wobj_Part_0;
        Movel Tr_meulage_bavure_102,VitesseRapide,Z0,Tool \Wobj:=Wobj_Part_0;
        Movel Tr_meulage_bavure_103,VitesseRapide,Z0,Tool \Wobj:=Wobj_Part_0;
        Movel Tr_meulage_bavure_104,VitesseRapide,Z0,Tool \Wobj:=Wobj_Part_0;
        Movel Tr_meulage_bavure_105,VitesseRapide,Z0,Tool \Wobj:=Wobj_Part_0;
        Movel Tr_meulage_bavure_106,VitesseRapide,Z0,Tool \Wobj:=Wobj_Part_0;
        Movel Tr_meulage_bavure_107,VitesseRapide,Z0,Tool \Wobj:=Wobj_Part_0;
        Movel Tr_meulage_bavure_108,VitesseRapide,Z0,Tool \Wobj:=Wobj_Part_0;
        Movel Tr_meulage_bavure_109,VitesseRapide,Z0,Tool \Wobj:=Wobj_Part_0;
        Movel Tr_meulage_bavure_110,VitesseRapide,Z0,Tool \Wobj:=Wobj_Part_0;
        Movel Tr_meulage_bavure_111,VitesseRapide,Z0,Tool \Wobj:=Wobj_Part_0;
        Movel Tr_meulage_bavure_112,VitesseRapide,Z0,Tool \Wobj:=Wobj_Part_0;
        Movel Tr_meulage_bavure_113,VitesseRapide,Z0,Tool \Wobj:=Wobj_Part_0;
        Movel Tr_meulage_bavure_114,VitesseRapide,Z0,Tool \Wobj:=Wobj_Part_0;
        Movel Tr_meulage_bavure_115,VitesseRapide,Z0,Tool \Wobj:=Wobj_Part_0;
        Movel Tr_meulage_bavure_116,VitesseRapide,Z0,Tool \Wobj:=Wobj_Part_0;
        Movel Tr_meulage_bavure_117,VitesseRapide,Z0,Tool \Wobj:=Wobj_Part_0;
        Movel Tr_meulage_bavure_118,VitesseRapide,Z0,Tool \Wobj:=Wobj_Part_0;
        Movel Tr_meulage_bavure_119,VitesseRapide,Z0,Tool \Wobj:=Wobj_Part_0;
        Movel Tr_meulage_bavure_120,VitesseRapide,Z0,Tool \Wobj:=Wobj_Part_0;
        Movel Tr_meulage_bavure_121,VitesseRapide,Z0,Tool \Wobj:=Wobj_Part_0;
        Movel Tr_meulage_bavure_122,VitesseRapide,Z0,Tool \Wobj:=Wobj_Part_0;
        Movel Tr_meulage_bavure_123,VitesseRapide,Z0,Tool \Wobj:=Wobj_Part_0;
        Movel Tr_meulage_bavure_124,VitesseRapide,Z0,Tool \Wobj:=Wobj_Part_0;
        Movel Tr_meulage_bavure_125,VitesseRapide,Z0,Tool \Wobj:=Wobj_Part_0;
        Movel Tr_meulage_bavure_126,VitesseRapide,Z0,Tool \Wobj:=Wobj_Part_0;
        Movel Tr_meulage_bavure_127,VitesseRapide,Z0,Tool \Wobj:=Wobj_Part_0;
        Movel Tr_meulage_bavure_128,VitesseRapide,Z0,Tool \Wobj:=Wobj_Part_0;
        Movel Tr_meulage_bavure_129,VitesseRapide,Z0,Tool \Wobj:=Wobj_Part_0;
        Movel Tr_meulage_bavure_130,VitesseRapide,Z0,Tool \Wobj:=Wobj_Part_0;
        Movel Tr_meulage_bavure_131,VitesseRapide,Z0,Tool \Wobj:=Wobj_Part_0;
        Movel Tr_meulage_bavure_132,VitesseRapide,Z0,Tool \Wobj:=Wobj_Part_0;
        Movel Tr_meulage_bavure_133,VitesseRapide,Z0,Tool \Wobj:=Wobj_Part_0;
        Movel Tr_meulage_bavure_134,VitesseRapide,Z0,Tool \Wobj:=Wobj_Part_0;
        Movel Tr_meulage_bavure_135,VitesseRapide,Z0,Tool \Wobj:=Wobj_Part_0;
        Movel Tr_meulage_bavure_136,VitesseRapide,Z0,Tool \Wobj:=Wobj_Part_0;
        Movel Tr_meulage_bavure_137,VitesseRapide,Z0,Tool \Wobj:=Wobj_Part_0;
        Movel Tr_meulage_bavure_138,VitesseRapide,Z0,Tool \Wobj:=Wobj_Part_0;
        Movel Tr_meulage_bavure_139,VitesseRapide,Z0,Tool \Wobj:=Wobj_Part_0;
        Movel Tr_meulage_bavure_140,VitesseRapide,Z0,Tool \Wobj:=Wobj_Part_0;
        Movel Tr_meulage_bavure_141,VitesseRapide,Z0,Tool \Wobj:=Wobj_Part_0;
        Movel Tr_meulage_bavure_142,VitesseRapide,Z0,Tool \Wobj:=Wobj_Part_0;
        Movel Tr_meulage_bavure_143,VitesseRapide,Z0,Tool \Wobj:=Wobj_Part_0;
        Movel Tr_meulage_bavure_144,VitesseRapide,Z0,Tool \Wobj:=Wobj_Part_0;
        Movel Tr_meulage_bavure_145,VitesseRapide,Z0,Tool \Wobj:=Wobj_Part_0;
        Movel Tr_meulage_bavure_146,VitesseRapide,Z0,Tool \Wobj:=Wobj_Part_0;
        Movel Tr_meulage_bavure_147,VitesseRapide,Z0,Tool \Wobj:=Wobj_Part_0;
        Movel Tr_meulage_bavure_148,VitesseRapide,Z0,Tool \Wobj:=Wobj_Part_0;
        Movel Tr_meulage_bavure_149,VitesseRapide,Z0,Tool \Wobj:=Wobj_Part_0;
        Movel Tr_meulage_bavure_150,VitesseRapide,Z0,Tool \Wobj:=Wobj_Part_0;
        Movel Tr_meulage_bavure_151,VitesseRapide,Z0,Tool \Wobj:=Wobj_Part_0;
        Movel Tr_meulage_bavure_152,VitesseRapide,Z0,Tool \Wobj:=Wobj_Part_0;
        Movel Tr_meulage_bavure_153,VitesseRapide,Z0,Tool \Wobj:=Wobj_Part_0;
        Movel Tr_meulage_bavure_154,VitesseRapide,Z0,Tool \Wobj:=Wobj_Part_0;
        Movel Tr_meulage_bavure_155,VitesseRapide,Z0,Tool \Wobj:=Wobj_Part_0;
        Movel Tr_meulage_bavure_156,VitesseRapide,Z0,Tool \Wobj:=Wobj_Part_0;
        Movel Tr_meulage_bavure_157,VitesseRapide,Z0,Tool \Wobj:=Wobj_Part_0;
        Movel Tr_meulage_bavure_158,VitesseRapide,Z0,Tool \Wobj:=Wobj_Part_0;
        Movel Tr_meulage_bavure_159,VitesseRapide,Z0,Tool \Wobj:=Wobj_Part_0;
        Movel Tr_meulage_bavure_160,VitesseRapide,Z0,Tool \Wobj:=Wobj_Part_0;
        Movel Tr_meulage_bavure_161,VitesseRapide,Z0,Tool \Wobj:=Wobj_Part_0;
        Movel Tr_meulage_bavure_162,VitesseRapide,Z0,Tool \Wobj:=Wobj_Part_0;
        Movel Tr_meulage_bavure_163,VitesseRapide,Z0,Tool \Wobj:=Wobj_Part_0;
        Movel Tr_meulage_bavure_164,VitesseRapide,Z0,Tool \Wobj:=Wobj_Part_0;
        Movel Tr_meulage_bavure_165,VitesseRapide,Z0,Tool \Wobj:=Wobj_Part_0;
        Movel Tr_meulage_bavure_166,VitesseRapide,Z0,Tool \Wobj:=Wobj_Part_0;
        Movel Tr_meulage_bavure_167,VitesseRapide,Z0,Tool \Wobj:=Wobj_Part_0;
        Movel Tr_meulage_bavure_168,VitesseRapide,Z0,Tool \Wobj:=Wobj_Part_0;
        Movel Tr_meulage_bavure_169,VitesseRapide,Z0,Tool \Wobj:=Wobj_Part_0;
        Movel Tr_meulage_bavure_170,VitesseRapide,Z0,Tool \Wobj:=Wobj_Part_0;
        Movel Tr_meulage_bavure_171,VitesseRapide,Z0,Tool \Wobj:=Wobj_Part_0;
        Movel Tr_meulage_bavure_172,VitesseRapide,Z0,Tool \Wobj:=Wobj_Part_0;
        Movel Tr_meulage_bavure_173,VitesseRapide,Z0,Tool \Wobj:=Wobj_Part_0;
        Movel Tr_meulage_bavure_174,VitesseRapide,Z0,Tool \Wobj:=Wobj_Part_0;
        Movel Tr_meulage_bavure_175,VitesseRapide,Z0,Tool \Wobj:=Wobj_Part_0;
        Movel Tr_meulage_bavure_176,VitesseRapide,Z0,Tool \Wobj:=Wobj_Part_0;
        Movel Tr_meulage_bavure_177,VitesseRapide,Z0,Tool \Wobj:=Wobj_Part_0;
        Movel Tr_meulage_bavure_178,VitesseLente,Z0,Tool \Wobj:=Wobj_Part_0;
        Movel Tr_meulage_bavure_179,VitesseLente,Z0,Tool \Wobj:=Wobj_Part_0;
        Movel Tr_meulage_bavure_180,VitesseLente,Z0,Tool \Wobj:=Wobj_Part_0;
        Movel Tr_meulage_bavure_181,VitesseLente,Z0,Tool \Wobj:=Wobj_Part_0;
        Movel Tr_meulage_bavure_182,VitesseLente,Z0,Tool \Wobj:=Wobj_Part_0;
        Movel Tr_meulage_bavure_183,VitesseLente,Z0,Tool \Wobj:=Wobj_Part_0;
        Movel Tr_meulage_bavure_184,VitesseLente,Z0,Tool \Wobj:=Wobj_Part_0;
        Movel Tr_meulage_bavure_185,VitesseLente,Z0,Tool \Wobj:=Wobj_Part_0;
        Movel Tr_meulage_bavure_186,VitesseLente,Z0,Tool \Wobj:=Wobj_Part_0;
        Movel Tr_meulage_bavure_187,VitesseLente,Z0,Tool \Wobj:=Wobj_Part_0;
        Movel Tr_meulage_bavure_188,VitesseLente,Z0,Tool \Wobj:=Wobj_Part_0;
        Movel Tr_meulage_bavure_189,VitesseLente,Z0,Tool \Wobj:=Wobj_Part_0;
        Movel Tr_meulage_bavure_190,VitesseLente,Z0,Tool \Wobj:=Wobj_Part_0;
        Movel Tr_meulage_bavure_191,VitesseLente,Z0,Tool \Wobj:=Wobj_Part_0;
        Movel Tr_meulage_bavure_192,VitesseLente,Z0,Tool \Wobj:=Wobj_Part_0;
        Movel Tr_meulage_bavure_193,VitesseLente,Z0,Tool \Wobj:=Wobj_Part_0;
        Movel Tr_meulage_bavure_194,VitesseLente,Z0,Tool \Wobj:=Wobj_Part_0;
        Movel Tr_meulage_bavure_195,VitesseLente,Z0,Tool \Wobj:=Wobj_Part_0;
        Movel Tr_meulage_bavure_196,VitesseLente,Z0,Tool \Wobj:=Wobj_Part_0;
        Movel Tr_meulage_bavure_197,VitesseLente,Z0,Tool \Wobj:=Wobj_Part_0;
        Movel Tr_meulage_bavure_198,VitesseLente,Z0,Tool \Wobj:=Wobj_Part_0;
        Movel Tr_meulage_bavure_199,VitesseLente,Z0,Tool \Wobj:=Wobj_Part_0;
        Movel Tr_meulage_bavure_200,VitesseLente,Z0,Tool \Wobj:=Wobj_Part_0;
        Movel Tr_meulage_bavure_201,VitesseLente,Z0,Tool \Wobj:=Wobj_Part_0;
        Movel Tr_meulage_bavure_202,VitesseLente,Z0,Tool \Wobj:=Wobj_Part_0;
        Movel Tr_meulage_bavure_203,VitesseLente,Z0,Tool \Wobj:=Wobj_Part_0;
        Movel Tr_meulage_bavure_204,VitesseLente,Z0,Tool \Wobj:=Wobj_Part_0;
        Movel Tr_meulage_bavure_205,VitesseLente,Z0,Tool \Wobj:=Wobj_Part_0;
        Movel Tr_meulage_bavure_206,VitesseLente,Z0,Tool \Wobj:=Wobj_Part_0;
        Movel Tr_meulage_bavure_207,VitesseLente,Z0,Tool \Wobj:=Wobj_Part_0;
        Movel Tr_meulage_bavure_208,VitesseLente,Z0,Tool \Wobj:=Wobj_Part_0;
        Movel Tr_meulage_bavure_209,VitesseLente,Z0,Tool \Wobj:=Wobj_Part_0;
        Movel Tr_meulage_bavure_210,VitesseRapide,Z0,Tool \Wobj:=Wobj_Part_0;
        Movel Tr_meulage_bavure_211,VitesseRapide,Z0,Tool \Wobj:=Wobj_Part_0;
        Movel Tr_meulage_bavure_212,VitesseRapide,Z0,Tool \Wobj:=Wobj_Part_0;
        Movel Tr_meulage_bavure_213,VitesseRapide,Z0,Tool \Wobj:=Wobj_Part_0;
        Movel Tr_meulage_bavure_214,VitesseRapide,Z0,Tool \Wobj:=Wobj_Part_0;
        Movel Tr_meulage_bavure_215,VitesseRapide,Z0,Tool \Wobj:=Wobj_Part_0;
        Movel Tr_meulage_bavure_216,VitesseRapide,Z0,Tool \Wobj:=Wobj_Part_0;
        Movel Tr_meulage_bavure_217,VitesseRapide,Z0,Tool \Wobj:=Wobj_Part_0;
        Movel Tr_meulage_bavure_218,VitesseRapide,Z0,Tool \Wobj:=Wobj_Part_0;
        Movel Tr_meulage_bavure_219,VitesseRapide,Z0,Tool \Wobj:=Wobj_Part_0;
        Movel Tr_meulage_bavure_220,VitesseRapide,Z0,Tool \Wobj:=Wobj_Part_0;
        Movel Tr_meulage_bavure_221,VitesseRapide,Z0,Tool \Wobj:=Wobj_Part_0;
        Movel Tr_meulage_bavure_222,VitesseRapide,Z0,Tool \Wobj:=Wobj_Part_0;
        Movel Tr_meulage_bavure_223,VitesseRapide,Z0,Tool \Wobj:=Wobj_Part_0;
        Movel Tr_meulage_bavure_224,VitesseRapide,Z0,Tool \Wobj:=Wobj_Part_0;
        Movel Tr_meulage_bavure_225,VitesseRapide,Z0,Tool \Wobj:=Wobj_Part_0;
        Movel Tr_meulage_bavure_226,VitesseRapide,Z0,Tool \Wobj:=Wobj_Part_0;
        Movel Tr_meulage_bavure_227,VitesseRapide,Z0,Tool \Wobj:=Wobj_Part_0;
        Movel Tr_meulage_bavure_228,VitesseRapide,Z0,Tool \Wobj:=Wobj_Part_0;
        Movel Tr_meulage_bavure_229,VitesseRapide,Z0,Tool \Wobj:=Wobj_Part_0;
        Movel Tr_meulage_bavure_230,VitesseRapide,Z0,Tool \Wobj:=Wobj_Part_0;
        Movel Tr_meulage_bavure_231,VitesseRapide,Z0,Tool \Wobj:=Wobj_Part_0;
        Movel Tr_meulage_bavure_232,VitesseRapide,Z0,Tool \Wobj:=Wobj_Part_0;
        Movel Tr_meulage_bavure_233,VitesseRapide,Z0,Tool \Wobj:=Wobj_Part_0;
        Movel Tr_meulage_bavure_234,VitesseRapide,Z0,Tool \Wobj:=Wobj_Part_0;
        Movel Tr_meulage_bavure_235,VitesseRapide,Z0,Tool \Wobj:=Wobj_Part_0;
        Movel Tr_meulage_bavure_236,VitesseRapide,Z0,Tool \Wobj:=Wobj_Part_0;
        Movel Tr_meulage_bavure_237,VitesseRapide,Z0,Tool \Wobj:=Wobj_Part_0;
        Movel Tr_meulage_bavure_238,VitesseRapide,Z0,Tool \Wobj:=Wobj_Part_0;
        Movel Tr_meulage_bavure_239,VitesseRapide,Z0,Tool \Wobj:=Wobj_Part_0;
        Movel Tr_meulage_bavure_240,VitesseRapide,Z0,Tool \Wobj:=Wobj_Part_0;
        Movel Tr_meulage_bavure_241,VitesseRapide,Z0,Tool \Wobj:=Wobj_Part_0;
        Movel Tr_meulage_bavure_242,VitesseRapide,Z0,Tool \Wobj:=Wobj_Part_0;
        Movel Tr_meulage_bavure_243,VitesseRapide,Z0,Tool \Wobj:=Wobj_Part_0;
        Movel Tr_meulage_bavure_244,VitesseRapide,Z0,Tool \Wobj:=Wobj_Part_0;
        Movel Tr_meulage_bavure_245,VitesseRapide,Z0,Tool \Wobj:=Wobj_Part_0;
        Movel Tr_meulage_bavure_246,VitesseRapide,Z0,Tool \Wobj:=Wobj_Part_0;
        Movel Tr_meulage_bavure_247,VitesseRapide,Z0,Tool \Wobj:=Wobj_Part_0;
        Movel Tr_meulage_bavure_248,VitesseRapide,Z0,Tool \Wobj:=Wobj_Part_0;
        Movel Tr_meulage_bavure_249,VitesseRapide,Z0,Tool \Wobj:=Wobj_Part_0;
        Movel Tr_meulage_bavure_250,VitesseRapide,Z0,Tool \Wobj:=Wobj_Part_0;
        Movel Tr_meulage_bavure_251,VitesseRapide,Z0,Tool \Wobj:=Wobj_Part_0;
        Movel Tr_meulage_bavure_252,VitesseRapide,Z0,Tool \Wobj:=Wobj_Part_0;
        Movel Tr_meulage_bavure_253,VitesseRapide,Z0,Tool \Wobj:=Wobj_Part_0;
        Movel Tr_meulage_bavure_254,VitesseRapide,Z0,Tool \Wobj:=Wobj_Part_0;
        Movel Tr_meulage_bavure_255,VitesseRapide,Z0,Tool \Wobj:=Wobj_Part_0;
        Movel Tr_meulage_bavure_256,VitesseRapide,Z0,Tool \Wobj:=Wobj_Part_0;
        Movel Tr_meulage_bavure_257,VitesseRapide,Z0,Tool \Wobj:=Wobj_Part_0;
        Movel Tr_meulage_bavure_258,VitesseRapide,Z0,Tool \Wobj:=Wobj_Part_0;
        Movel Tr_meulage_bavure_259,VitesseRapide,Z0,Tool \Wobj:=Wobj_Part_0;
        Movel Tr_meulage_bavure_260,VitesseRapide,Z0,Tool \Wobj:=Wobj_Part_0;
        Movel Tr_meulage_bavure_261,VitesseRapide,Z0,Tool \Wobj:=Wobj_Part_0;
        Movel Tr_meulage_bavure_262,VitesseRapide,Z0,Tool \Wobj:=Wobj_Part_0;
        Movel Tr_meulage_bavure_263,VitesseRapide,Z0,Tool \Wobj:=Wobj_Part_0;
        Movel Tr_meulage_bavure_264,VitesseRapide,Z0,Tool \Wobj:=Wobj_Part_0;
        Movel Tr_meulage_bavure_265,VitesseRapide,Z0,Tool \Wobj:=Wobj_Part_0;
        Movel Tr_meulage_bavure_266,VitesseRapide,Z0,Tool \Wobj:=Wobj_Part_0;
        Movel Tr_meulage_bavure_267,VitesseRapide,Z0,Tool \Wobj:=Wobj_Part_0;
        Movel Tr_meulage_bavure_268,VitesseRapide,Z0,Tool \Wobj:=Wobj_Part_0;
        Movel Tr_meulage_bavure_269,VitesseRapide,Z0,Tool \Wobj:=Wobj_Part_0;
        Movel Tr_meulage_bavure_270,VitesseRapide,Z0,Tool \Wobj:=Wobj_Part_0;
        Movel Tr_meulage_bavure_271,VitesseRapide,Z0,Tool \Wobj:=Wobj_Part_0;
        Movel Tr_meulage_bavure_272,VitesseRapide,Z0,Tool \Wobj:=Wobj_Part_0;
        Movel Tr_meulage_bavure_273,VitesseRapide,Z0,Tool \Wobj:=Wobj_Part_0;
        Movel Tr_meulage_bavure_274,VitesseRapide,Z0,Tool \Wobj:=Wobj_Part_0;
        Movel Tr_meulage_bavure_275,VitesseRapide,Z0,Tool \Wobj:=Wobj_Part_0;
        Movel Tr_meulage_bavure_276,VitesseRapide,Z0,Tool \Wobj:=Wobj_Part_0;
        Movel Tr_meulage_bavure_277,VitesseRapide,Z0,Tool \Wobj:=Wobj_Part_0;
        Movel Tr_meulage_bavure_278,VitesseRapide,Z0,Tool \Wobj:=Wobj_Part_0;
        Movel Tr_meulage_bavure_279,VitesseRapide,Z0,Tool \Wobj:=Wobj_Part_0;
        Movel Tr_meulage_bavure_280,VitesseRapide,Z0,Tool \Wobj:=Wobj_Part_0;
        Movel Tr_meulage_bavure_281,VitesseRapide,Z0,Tool \Wobj:=Wobj_Part_0;
        Movel Tr_meulage_bavure_282,VitesseRapide,Z0,Tool \Wobj:=Wobj_Part_0;
        Movel Tr_meulage_bavure_283,VitesseRapide,Z0,Tool \Wobj:=Wobj_Part_0;
        Movel Tr_meulage_bavure_284,VitesseRapide,Z0,Tool \Wobj:=Wobj_Part_0;
        Movel Tr_meulage_bavure_285,VitesseRapide,Z0,Tool \Wobj:=Wobj_Part_0;
        Movel Tr_meulage_bavure_286,VitesseRapide,Z0,Tool \Wobj:=Wobj_Part_0;
        Movel Tr_meulage_bavure_287,VitesseRapide,Z0,Tool \Wobj:=Wobj_Part_0;
        Movel Tr_meulage_bavure_288,VitesseRapide,Z0,Tool \Wobj:=Wobj_Part_0;
        Movel Tr_meulage_bavure_289,VitesseRapide,Z0,Tool \Wobj:=Wobj_Part_0;
        Movel Tr_meulage_bavure_290,VitesseRapide,Z0,Tool \Wobj:=Wobj_Part_0;
        Movel Tr_meulage_bavure_291,VitesseRapide,Z0,Tool \Wobj:=Wobj_Part_0;
        Movel Tr_meulage_bavure_292,VitesseRapide,Z0,Tool \Wobj:=Wobj_Part_0;
        Movel Tr_meulage_bavure_293,VitesseRapide,Z0,Tool \Wobj:=Wobj_Part_0;
        Movel Tr_meulage_bavure_294,VitesseRapide,Z0,Tool \Wobj:=Wobj_Part_0;
        Movel Tr_meulage_bavure_295,VitesseRapide,Z0,Tool \Wobj:=Wobj_Part_0;
        Movel Tr_meulage_bavure_296,VitesseRapide,Z0,Tool \Wobj:=Wobj_Part_0;
        !
        !Degagement
        MoveL Reltool(Tr_meulage_bavure_296,0,0,-10),V100,Z0,Tool \Wobj:=Wobj_Part_0;
        MoveL Reltool(Tr_meulage_bavure_296,0,0,-100),V500,Z0,Tool \Wobj:=Wobj_Part_0;
        MoveJ Reltool(Tr_meulage_bavure_296,0,0,-200),V1000,Z0,Tool \Wobj:=Wobj_Part_0;


        Go_to_Meulage_Plan;
        !
        !

    ENDPROC

    !Trajectoire de depose de la piece
    LOCAL PROC DEPOSE()
        !
        stop;

        PEO;

        !
        !Approche
		MoveJ Reltool(PicKPosition,0,0,-200),V1000,Z0,Tool_Prehenseur1 \Wobj:=Wobj_vision;
		MoveL Reltool(PicKPosition,0,0,-100),V500,Z0,Tool_Prehenseur1 \Wobj:=Wobj_vision;
		MoveL Reltool(PicKPosition,0,0,-10),V200,Z0,Tool_Prehenseur1 \Wobj:=Wobj_vision;
		MoveL PicKPosition,V100,Fine,Tool_Prehenseur1 \Wobj:=Wobj_vision;

        !Fermeture pince
		Gripper_Open;
        !
		MoveL Reltool(PicKPosition,0,0,-200),V500,Z0,Tool_Prehenseur1 \Wobj:=Wobj_vision;

        !
        PEO;
        !

        !Gripper_Close;

        !
    ENDPROC

ENDMODULE
